Staubli VAL3: OnF6.pgx

public program OnF6()
begin
end
